TYPE Tc2_EtherCAT_Error_typ :
	STRUCT
		ErrorID : UDINT ;
		ErrorText : STRING[2048];
	END_STRUCT
END_TYPE

(* stored: Version 1.1.0.1, ProductVersion 3.1.4024.3
   DUT Tc2_EtherCAT_Error_typ: Id {90066b92-a65a-0812-06d1-2b16b93a1276} *)
